(* IEC 61131-3 sources: PLC/exercises, 9 files *)

(* ---- practice_10.st ---- *)
(*
 * non revisonato
**)

PROGRAM _INIT

END_PROGRAM

PROGRAM _CYCLIC

    VAR
        start_button := "ingresso_1";
        stop_button := "ingresso_2";
        sensore_imbuto_alto := "ingresso_3";                 // Sensore parte alta dell'imbuto
        sensore_imbuto_basso := "ingresso_4";                // Sensore parte bassa dell'imbuto

        "uscita_1" := cilindro_valvola_ingersso_imbuto;      // Per rempimento imbuto
        "uscita_2" := cilindro_valvola_uscita_imbuto;        // Per svutamento imbuto
        "uscita_2" := motore_nasto_trasportatore;
        "uscita_2" := forno_cottura;

    END_VAR

    IF start_button AND NOT stop_button THEN
        start_ciclo.sensore_imbuto_basso := sensore_imbuto_basso;
        start_ciclo.sensore_imbuto_basso := sensore_imbuto_basso;
        start_ciclo.cilindro_valvola_ingersso_imbuto := cilindro_valvola_uscita_imbuto;
        start_ciclo.cilindro_valvola_uscita_imbuto := cilindro_valvola_uscita_imbuto;
        start_ciclo.motore_nasto_trasportatore := motore_nasto_trasportatore;
        start_ciclo.forno_cottura := forno_cottura;
        start_ciclo();
    ELSIF stop_button AND NOT start_button THEN
        stop_ciclo.cilindro_valvola_ingersso_imbuto := cilindro_valvola_uscita_imbuto;
        stop_ciclo.cilindro_valvola_uscita_imbuto := cilindro_valvola_uscita_imbuto;
        stop_ciclo.motore_nasto_trasportatore := motore_nasto_trasportatore;
        stop_ciclo.forno_cottura := forno_cottura;
        stop_ciclo();
    END_IF;

    FUNCTION_BLOCK start_ciclo
        (*
         * Avvia il ciclo produttivo del forno
        **)
        VAR_INPUT
            sensore_imbuto_alto: BOOL;
            sensore_imbuto_basso: BOOL;

            cilindro_valvola_ingersso_imbuto: BOOL;
            cilindro_valvola_uscita_imbuto: BOOL;
            motore_nasto_trasportatore: BOOL;
            forno_cottura: BOOL;
        END_VAR
        VAR
            fase := 0;
            timer_nastro := 0;
            timer_forno := 0;
        END_VAR

        IF sistem_bit_1sec AND motore_nasto_trasportatore THEN
            timer_nastro := timer_nastro + 1;
        ELSIF sistem_bit_1sec AND forno_cottura THEN
            timer_forno := timer_forno + 1;
        END_IF;

        CASE fase OF
            0:
                (*
                 * Controllo riempimento/svuotamento imbuto
                 *
                 * Entry point
                **)
                IF NOT sensore_imbuto_alto AND NOT sensore_imbuto_basso THEN
                    cilindro_valvola_uscita_imbuto := 0;
                    cilindro_valvola_ingersso_imbuto := 1;
                ELSIF sensore_imbuto_alto AND sensore_imbuto_basso THEN
                    cilindro_valvola_ingersso_imbuto := 0;
                    cilindro_valvola_uscita_imbuto := 1;
                    fase := 10;
                END_IF;

            10:
                (*
                 * Avvio e arresto nastro trasportatore per ingresso forno
                 *
                 * Entrata → fase 0 (riempimento/svuotamento imbuto)
                 * Uscita → fase 20 (forno cottura)
                **)
                IF NOT motore_nasto_trasportatore AND timer_nastro == 0 THEN
                    motore_nasto_trasportatore := 1;
                ELSIF motore_nasto_trasportatore AND timer_nastro == 15 THEN
                    motore_nasto_trasportatore := 0;
                    timer_nastro := 0;
                    fase := 20;
                END_IF;

            20:
                (*
                 * Accensione e spegnimento forno cottura
                 *
                 * Entrata → fase 20 (nastro trasportatore per ingresso forno)
                 * Uscita → fase 30 (nastro trasportatore per uscita forno)
                **)
                IF NOT forno_cottura THEN
                    forno_cottura := 1;
                ELSIF forno_cottura AND timer_forno == 10 THEN
                    forno_cottura := 0;
                    timer_forno := 0;
                    fase := 30;
                END_IF;

            30:
                (*
                 * Avvio e arresto nastro trasportatore per uscita forno
                 *
                 * Entrata → fase 30 (forno cottura)
                 * Uscita → fase 0 (riempimento/svuotamento imbuto)
                **)
                IF NOT motore_nasto_trasportatore THEN
                    motore_nasto_trasportatore := 1;
                ELSIF motore_nasto_trasportatore AND timer_nastro == 10 THEN
                    motore_nasto_trasportatore := 0;
                    timer_nastro := 0;
                    fase := 0;
                END_IF;

        END_CASE;

    END_FUNCTION_BLOCK

    FUNCTION_BLOCK stop_ciclo
        (*
         * Ferma il ciclo produttivo del forno
        **)
        VAR_INPUT
            cilindro_valvola_ingersso_imbuto: BOOL;
            cilindro_valvola_uscita_imbuto: BOOL;
            motore_nasto_trasportatore: BOOL;
            forno_cottura: BOOL;
        END_VAR

            cilindro_valvola_ingersso_imbuto := 0;
            cilindro_valvola_uscita_imbuto := 0;
            motore_nasto_trasportatore =: 0;
            forno_cottura := 0;

    END_FUNCTION_BLOCK

END_PROGRAM

PROGRAM _EXIT

END_PROGRAM

(* ---- practice_14.st ---- *)
(*
 * non revisionato
**)

PROGRAM _INIT

END_PROGRAM

PROGRAM _CYCLIC

    VAR
        A := "ingresso_1";
        B := "ingresso_2";
        conteggio : INT := 0;
    END_VAR

    contatore.A := A;
    contatore.B := B;
    contatore.conteggio := conteggio;
    contatore();

    FUNCTION_BLOCK contatore
        VAR_INPUT
            A : BOOL;
            B : BOOL;
            conteggio : INT;
        END_VAR
        VAR
            orario: BOOL := 0;
        END_VAR

        CASE fase OF
        0:
            IF NOT A AND NOT B THEN
                fase := 10;
            END_IF;
        10:
            IF A XOR B THEN
                IF A AND NOT B THEN
                    orario := 1;
                ELSIF NOT A AND B THEN
                    orario := 0;
                END_IF;
                fase := 20;
            END_IF;
        20:
            IF A AND B THEN
                fase := 30;
            END_IF;
        30:
            IF A XOR B THEN
                fase := 40;
            END_IF;
        40:
            IF orario THEN
                conteggio := conteggio + 1;
            ELSE
                conteggio := conteggio - 1;
            END_IF;
            fase := 0;

    END_FUNCTION_BLOCK

END_PROGRAM

PROGRAM _EXIT

END_PROGRAM

(* ---- practice_15.st ---- *)
(*
 * non revisionato
**)

PROGRAM _INIT

END_PROGRAM

PROGRAM _CYCLIC

    VAR
        A := "ingresso_1";
        B := "ingresso_2";
        preset := "ingresso_3";
        conteggio : INT := 0;
        orario: BOOL := 0;
        "uscita_4" := trasporto;
    END_VAR

    contatore.A := A;
    contatore.B := B;
    contatore.conteggio := conteggio;
    contatore();

    IF preset THEN
        contatore.conteggio := 0;
    END_IF;

    IF contatore.conteggio MOD 1000 == 0 THEN
        trasporto := 1;
    END_IF;

    FUNCTION_BLOCK contatore
        VAR_INPUT
            A : BOOL;
            B : BOOL;
            conteggio : INT;
        END_VAR
        VAR
            orario: BOOL := 0;
        END_VAR

        CASE fase OF
        0:
            IF NOT A AND NOT B THEN
                fase := 10;
            END_IF;
        10:
            IF A XOR B THEN
                IF A AND NOT B THEN
                    orario := 1;
                ELSIF NOT A AND B THEN
                    orario := 0;
                END_IF;
                fase := 20;
            END_IF;
        20:
            IF A AND B THEN
                fase := 30;
            END_IF;
        30:
            IF A XOR B THEN
                fase := 40;
            END_IF;
        40:
            IF orario THEN
                conteggio := conteggio + 1;
            ELSE
                conteggio := conteggio - 1;
            END_IF;
            fase := 0;

    END_FUNCTION_BLOCK

END_PROGRAM

PROGRAM _EXIT

END_PROGRAM

(* ---- practice_16.st ---- *)
(*
 * non revisionato
**)

PROGRAM _INIT

END_PROGRAM

PROGRAM _CYCLIC

    VAR
        A := "ingresso_1";
        B := "ingresso_2";
        reset := "ingresso_3";

        conteggio : INT := 0;

        "uscita_1" := led[0];
        "uscita_2" := led[1];
        "uscita_3" := led[2];
        "uscita_4" := led[3];
        "uscita_5" := led[4];
        "uscita_6" := led[5];
        "uscita_7" := led[6];
        "uscita_8" := led[7];
        "uscita_9" := led[8];
        "uscita_10" := led[9];
    END_VAR

    contatore.A := A;
    contatore.B := B;
    contatore.conteggio := conteggio;
    contatore();

    IF contatore.conteggio MOD 100 THEN
        FOR x := 0 TO conteggio BY 100 DO
            led[x] := 0;
        END_FOR;
    END_IF;

    IF reset OR contatore.conteggio MOD 2000 == 0 THEN
        FOR x := 0 TO 9 DO
           led[x] := 0;
        END_FOR;
    END_IF;

    FUNCTION_BLOCK contatore
        VAR_INPUT
            A : BOOL;
            B : BOOL;
            conteggio : INT;
        END_VAR
        VAR
            orario: BOOL := 0;
        END_VAR

        CASE fase OF
        0:
            IF NOT A AND NOT B THEN
                fase := 10;
            END_IF;
        10:
            IF A XOR B THEN
                IF A AND NOT B THEN
                    orario := 1;
                ELSIF NOT A AND B THEN
                    orario := 0;
                END_IF;
                fase := 20;
            END_IF;
        20:
            IF A AND B THEN
                fase := 30;
            END_IF;
        30:
            IF A XOR B THEN
                fase := 40;
            END_IF;
        40:
            IF orario THEN
                conteggio := conteggio + 1;
            ELSE
                conteggio := conteggio - 1;
            END_IF;
            fase := 0;

    END_FUNCTION_BLOCK

END_PROGRAM

PROGRAM _EXIT

END_PROGRAM

(* ---- practice_01.st ---- *)
(*
    EXERCISE 01

    Author: Chiliano Arcarese
    Revised by IVAN
*)

PROGRAM _INIT

END_PROGRAM

PROGRAM _CYCLIC

    VAR
        ingresso_rele := "ingresso_1";
        "uscita_1" := uscita_motore;
    END_VAR

    IF ingresso_rele AND uscita_motore THEN
        uscita_motore := 0;
    END_IF;

END_PROGRAM

PROGRAM _EXIT

END_PROGRAM

(* ---- practice_09.st ---- *)
(*
 * es 09
 * revisionato.
**)

PROGRAM _INIT
END_PROGRAM

PROGRAM _CYCLIC

    VAR

        (*
         *  >>>>>>>>>>>>>> !-NOTA-BENE-! <<<<<<<<<<<<<<<
         *
         *  I PIANI SONO NOMINATI COME 1°, 2° E 3.
         *  IL PIANO TERRA CORRISPONDE AL 1° PIANO.
         *
         *  >>>>>>>>>>>>>> !-NOTA-BENE-! <<<<<<<<<<<<<<<
        **)

        // Contesto relativo al 1 piano dell'edificio
        "uscita_1" := led_piano_1;                       // LED di segnalazione movimento cabina (1 == movimento)
        pulsante_chiamata_piano_1 := "ingresso_1";       // Pulsante di chiamata della cabina
        sensore_arrivo_piano_1 := "ingresso_2";          // Sensore di arrivo della cabina (1 == cabina presente)

        // Contesto relativo al 2 piano dell'edificio
        "uscita_2" := led_piano_2;
        pulsante_chiamata_piano_2 := "ingresso_3";
        sensore_arrivo_piano_2 := "ingresso_4";

        // Contesto relativo al 3 piano dell'edificio
        "uscita_3" := led_piano_3;
        pulsante_chiamata_piano_3 := "ingresso_5";
        sensore_arrivo_piano_3 := "ingresso_6";

        // Contesto interno alla cabina dell'ascensore
        pulsante_cabina_piano_1 := "ingresso_7";           //
        pulsante_cabina_piano_2 := "ingresso_8";           // Pulsante destinazione cabina
        pulsante_cabina_piano_3 := "ingresso_9";           //
        sensore_chiusura_porte := "ingresso_10";           // Sensore chiusura porte (1 == chiuse)
        pulsante_allarme := "ingresso_11";                 // Pulsante di emergenza, attiva un allarme di 20s
        allarme_cabina := "uscita_8";

        // Contesto motori cabina
        "uscita_4" := motore_up;
        "uscita_5" := motore_down;

        // Contesto motori porte
        "uscita_6" := motore_porte_open;
        "uscita_7" := motore_porte_close;

        timer: INT := 0;
        timer_porta: INT := 0;

    END_VAR

    (*
     * Inizializzazione variabili funzione `movimento_cabina`
    **)
    // Led movimento cabina
    movimento_cabina.led_piano_1 := led_piano_1;
    movimento_cabina.led_piano_2 := led_piano_2;
    movimento_cabina.led_piano_3 := led_piano_3;
    // Sensori presenza cabina
    movimento_cabina.sensore_arrivo_piano_1 := sensore_arrivo_piano_1;
    movimento_cabina.sensore_arrivo_piano_2 := sensore_arrivo_piano_2;
    movimento_cabina.sensore_arrivo_piano_3 := sensore_arrivo_piano_3;
     // Porte cabina
    movimento_cabina.sensore_chiusura_porte := sensore_chiusura_porte;
    movimento_cabina.motore_porte_open := motore_porte_open;
    // Motori cabina
    movimento_cabina.motore_up := motore_up;
    movimento_cabina.motore_down := motore_down;

    (*
     * Chiamata della cabina da uno dei piani presenti.
    **)
    IF pulsante_chiamata_piano_1 THEN
        movimento_cabina.chiamta_esterna := TRUE;
        movimento_cabina.pulsante_chiamata := pulsante_chiamata_piano_1;
        movimento_cabina.piano_chiamata := 1;
        movimento_cabina();
    ELSIF pulsante_chiamata_piano_2 THEN
        movimento_cabina.chiamta_esterna := TRUE;
        movimento_cabina.pulsante_chiamata := pulsante_chiamata_piano_2;
        movimento_cabina.piano_chiamata := 2;
        movimento_cabina();
    ELSIF pulsante_chiamata_piano_3 THEN
        movimento_cabina.chiamta_esterna := TRUE;
        movimento_cabina.pulsante_chiamata := pulsante_chiamata_piano_3;
        movimento_cabina.piano_chiamata := 3;
        movimento_cabina();
    END_IF;

    (*
     * Risposta della cabina da pulsante interno.
    **)
    IF pulsante_cabina_piano_1 AND NOT sensore_arrivo_piano_1 THEN
        movimento_cabina.chiamta_esterna := FALSE;
        movimento_cabina.pulsante_chiamata := pulsante_cabina_piano_1;
        movimento_cabina.piano_chiamata := 1;
        movimento_cabina();
    ELSIF pulsante_cabina_piano_2 AND NOT sensore_arrivo_piano_2 THEN
        movimento_cabina.chiamta_esterna := FALSE;
        movimento_cabina.pulsante_chiamata := pulsante_cabina_piano_2;
        movimento_cabina.piano_chiamata := 2;
        movimento_cabina();
    ELSIF pulsante_cabina_piano_3 AND NOT sensore_arrivo_piano_3 THEN
        movimento_cabina.chiamta_esterna := FALSE;
        movimento_cabina.pulsante_chiamata := pulsante_cabina_piano_3;
        movimento_cabina.piano_chiamata := 3;
        movimento_cabina();
    END_IF;

    IF pulsante_allarme THEN
        allarme_cabina := 1;
        timer := 0;
    END_IF;

    IF sistem_bit_1sec THEN
        timer := timer + 1;
    END_IF;

    IF sistem_bit_1sec AND NOT sensore_chiusura_porte THEN
        timer_porta := timer_porta + 1;
    END_IF;

    IF timer == 20 AND allarme_cabina THEN
        allarme_cabina := 0;
        timer := 0;
    END_IF;

    // Chiusura porta ascensore automatica dopo 40 sec
    IF timer_porta > 40 AND NOT sensore_chiusura_porte AND NOT motore_porte_close THEN
        timer_porta := 0;
        motore_porte_close := 1;
    ELSIF sensore_chiusura_porte AND motore_porte_close THEN
        motore_porte_close := 0;
    END_IF;
 THEN

    FUNCTION_BLOCK movimento_cabina
    (*
     * Muove la cabina sui piani in base agli input dei pulsanti presenti in ogni piano.
    **)

        VAR_INPUT
            piano_chiamata: INT;
            chiamta_esterna: BOOL;
            pulsante_chiamata: BOOL;            // Pulsante di chiamata della cabina
            led_piano_1: BOOL;
            led_piano_2: BOOL;
            led_piano_3: BOOL;

            // Sensori presenza cabina
            sensore_arrivo_piano_1: BOOL;
            sensore_arrivo_piano_2: BOOL;
            sensore_arrivo_piano_3: BOOL;

            // Porte cabina
            sensore_chiusura_porte: BOOL;
            motore_porte_open: BOOL;

            // Motori cabina
            motore_up: BOOL;
            motore_down: BOOL;
        END_VAR

        VAR
            fase: INT := 0;                     // Variabile locale per i casi del CASE OF
        END_VAR

        IF pulsante_chiamata_piano AND NOT led_piano_1 AND NOT led_piano_2 AND NOT led_piano_3 THEN
            // Segnalo cabina in uso su tutti i piani
            led_piano_1 := TRUE;
            led_piano_2 := TRUE;
            led_piano_3 := TRUE;

            CASE fase OF

                0:
                    (*
                     * Localizzazione della cabina fra i piani e reindirizzamento verso il piano di chiamata.
                     *
                     * Entrate → Case entry point
                     *
                     * Uscite  → Spostamenti cabina (30, 40, 50)
                     *           Apertura porte (10)
                    **)
                    IF sensore_arrivo_piano_1 AND NOT sensore_arrivo_piano_2 AND NOT sensore_arrivo_piano_3 THEN
                        // Chiamata da piano
                        IF piano_chiamata == 1 AND chiamta_esterna THEN
                            fase := 10;
                        ELSIF piano_chiamata == 2 AND chiamta_esterna THEN
                            fase := 50;
                        ELSIF piano_chiamata == 3 AND chiamta_esterna THEN
                            fase := 40;
                        // Chiamata da cabina
                        ELSIF piano_chiamata == 1 AND NOT chiamta_esterna THEN
                            fase := 0;
                        ELSIF piano_chiamata == 2 AND NOT chiamta_esterna THEN
                            fase := 20;
                        ELSIF piano_chiamata == 3 AND NOT chiamta_esterna THEN
                            fase := 20;
                        END_IF;
                    ELSIF NOT sensore_arrivo_piano_1 AND sensore_arrivo_piano_2 AND NOT sensore_arrivo_piano_3 THEN
                        // Chiamata da piano
                        IF piano_chiamata == 1 AND chiamta_esterna THEN
                            fase := 30;
                        ELSIF piano_chiamata == 2 AND chiamta_esterna THEN
                            fase := 10;
                        ELSIF piano_chiamata == 3 AND chiamta_esterna THEN
                            fase := 40;
                        // Chiamata da cabina
                        ELSIF piano_chiamata == 1 AND NOT chiamta_esterna THEN
                            fase := 0;
                        ELSIF piano_chiamata == 2 AND NOT chiamta_esterna THEN
                            fase := 20;
                        ELSIF piano_chiamata == 3 AND NOT chiamta_esterna THEN
                            fase := 20;
                        END_IF;
                    ELSIF NOT sensore_arrivo_piano_1 AND NOT sensore_arrivo_piano_2 AND sensore_arrivo_piano_3 THEN
                        // Chiamata da piano
                        IF piano_chiamata == 1 AND chiamta_esterna THEN
                            fase := 30;
                        ELSIF piano_chiamata == 2 AND chiamta_esterna THEN
                            fase := 50;
                        ELSIF piano_chiamata == 3 AND chiamta_esterna THEN
                            fase := 10;
                        // Chiamata da cabina
                        ELSIF piano_chiamata == 1 AND NOT chiamta_esterna THEN
                            fase := 0;
                        ELSIF piano_chiamata == 2 AND NOT chiamta_esterna THEN
                            fase := 20;
                        ELSIF piano_chiamata == 3 AND NOT chiamta_esterna THEN
                            fase := 20;
                        END_IF;
                    END_IF;

                10:
                    (*
                     * Apertura porte cabina.
                     *
                     * Entrata → Localizzazione e reindirizzamento (0)
                    **)
                    IF sensore_chiusura_porte AND NOT motore_porte_open THEN
                        motore_porte_open := 1;
                    ELSIF NOT sensore_chiusura_porte AND motore_porte_open THEN
                        motore_porte_open := 0;
                    END_IF;
                    fase := 0;

                20:
                    (*
                     * Chiusura porte cabina.
                     *
                     * Entrata → Localizzazione e reindirizzamento (0)
                    **)
                    IF NOT sensore_chiusura_porte AND NOT motore_porte_close THEN
                        motore_porte_close := 1;
                    ELSIF sensore_chiusura_porte AND motore_porte_close THEN
                        motore_porte_close := 0;
                    END_IF;
                    fase := 0;
                    // In fase 0 il movimento viene poi gestito come una chiamata a piano ma pertendo a porte chiuse
                    chiamta_esterna := TRUE;

                30:
                    (*
                     * Spostamento cabina verso il 1° piano.
                     *
                     * Entrata → Localizzazione e reindirizzamento (0)
                     *
                     * Uscita → Apertura porte (10)
                    **)
                    IF NOT motore_up AND NOT motore_down AND sensore_chiusura_porte THEN
                        motore_down := 1;
                    ELSIF NOT motore_up AND motore_down AND sensore_arrivo_piano_1 THEN
                        motore_down := 0;
                        fase := 10;
                    ELSIF motore_up OR motore_down AND NOT sensore_chiusura_porte THEN
                        // ALLARME PORTA CABINA APERTA
                    END_IF;

                40:
                    (*
                     * Spostamento cabina verso il 3° piano.
                     *
                     * Entrata → Localizzazione e reindirizzamento (0)
                     *
                     * Uscita → Apertura porte (10)
                    **)
                    IF NOT motore_up AND NOT motore_down AND sensore_chiusura_porte THEN
                        motore_up := 1;
                    ELSIF motore_up AND NOT motore_down AND sensore_arrivo_piano_3 THEN
                        motore_up := 0;
                        fase := 10;
                    ELSIF motore_up OR motore_down AND NOT sensore_chiusura_porte THEN
                        // ALLARME PORTA CABINA APERTA
                    END_IF;

                50:
                    (*
                     * Spostamento cabina verso il 2° piano. La cabina si sporterà a partire dal basso o dall'alto.
                     *
                     * Entrata → Localizzazione e reindirizzamento (0)
                     *
                     * Uscita → Apertura porte (10)
                    **)
                    IF NOT motore_up AND NOT motore_down THEN
                        IF sensore_arrivo_piano_3 AND NOT sensore_arrivo_piano_1 AND NOT sensore_arrivo_piano_2 THEN
                            motore_down := 1;
                        ELSIF sensore_arrivo_piano_1 AND NOT sensore_arrivo_piano_2 AND NOT sensore_arrivo_piano_3 THEN
                            motore_up := 1;
                        END_IF;
                    ELSIF motore_down AND NOT motore_up THEN
                        IF sensore_arrivo_piano_2 THEN
                            motore_down := 0;
                            fase := 10;
                        END_IF;
                    ELSIF NOT motore_down AND motore_up THEN
                        IF sensore_arrivo_piano_2 THEN
                            motore_up := 0;
                            fase := 10;
                        END_IF;

            END_CASE;

        END_IF;

    END_FUNCTION_BLOCK

END_PROGRAM

PROGRAM _EXIT
END_PROGRAM

(* ---- practice_11.st ---- *)
(*
 * non revisionato
**)

PROGRAM _INIT

END_PROGRAM

PROGRAM _CYCLIC

    VAR
        rele[0] := "ingresso_1"
        rele[1] := "ingresso_2"
        rele[2] := "ingresso_3"
        rele[3] := "ingresso_4"
        rele[4] := "ingresso_5"
        rele[6] := "ingresso_6"
        rele[7] := "ingresso_7"
        rele[8] := "ingresso_8"
        rele[9] := "ingresso_9"
        rele[10] := "ingresso_10"

        "uscita_1" := motori[0];
        "uscita_2" := motori[1];
        "uscita_3" := motori[2];
        "uscita_4" := motori[3];
        "uscita_5" := motori[4];
        "uscita_6" := motori[5];
        "uscita_7" := motori[6];
        "uscita_8" := motori[7];
        "uscita_9" := motori[8];
        "uscita_10" := motori[9];
    END_VAR

    FOR x := 0 TO 9 BY 1 DO
        IF rele[0] THEN
            motori[x] := 0;
        ELSE
            motori[x] := 1;
        END_IF;
    END_FOR;

END_PROGRAM

PROGRAM _EXIT

END_PROGRAM

(* ---- practice_12.st ---- *)
(*
 * non revisionato
**)

PROGRAM _INIT

END_PROGRAM

PROGRAM _CYCLIC

    VAR
        pulsante := "ingresso_1";
        "uscita_1" := led[0]
        "uscita_2" := led[1]
        "uscita_3" := led[2]
        "uscita_4" := led[3]
        "uscita_5" := led[4]
        "uscita_6" := led[5]
        "uscita_7" := led[6]
        "uscita_8" := led[7]
        "uscita_9" := led[8]
        "uscita_10" := led[9]
        fase : INT := 0;
    END_VAR

    IF pulsante THEN
        CASE fase OF
            0:
                led[fase] := 1;
                fase := fase + 1;
            1:
                led[fase] := 1;
                fase := fase + 1;
            2:
                led[fase] := 1;
                fase := fase + 1;
            3:
                led[fase] := 1;
                fase := fase + 1;
            4:
                led[fase] := 1;
                fase := fase + 1;
            5:
                led[fase] := 1;
                fase := fase + 1;
            6:
                led[fase] := 1;
                fase := fase + 1;
            7:
                led[fase] := 1;
                fase := fase + 1;
            8:
                led[fase] := 1;
                fase := fase + 1;
            9:
                led[fase] := 1;
                fase := fase + 1;
            10:
                FOR x := 0 TO 9 DO
                    led[x] := 0;
                END_FOR;
                fase := 0;

        END_CASE;

END_PROGRAM

PROGRAM _EXIT

END_PROGRAM

(* ---- practice_17.st ---- *)
(*
 * non revisionato
**)

PROGRAM _INIT

END_PROGRAM

PROGRAM _CYCLIC

    VAR
        pulsante_carico_ricetta := "ingresso_1";
        finecorsa_passo         := "ingresso_2";
        ricetta : ARRAY[0..10]  := "ingresso_3";

        nr_posizione : INT := 0;
        posizione;
        appoggio1;
        appoggio2;

        mappa : ARRAY[0..10] OF ARRAY[1..10] := [
            pos_1 : ARRAY[0..10] OF INT, pos_2 : ARRAY[0..10] OF INT, pos_3 : ARRAY[0..10] OF INT,
            pos_4 : ARRAY[0..10] OF INT, pos_5 : ARRAY[0..10] OF INT, pos_6 : ARRAY[0..10] OF INT,
            pos_7 : ARRAY[0..10] OF INT, pos_8 : ARRAY[0..10] OF INT, pos_9 : ARRAY[0..10] OF INT,
            pos_10 : ARRAY[0..10] OF INT
        ];
    END_VAR

    IF nr_posizione >= 10 THEN
        nr_posizione := 0;
    END_IF;

    prima_colonna_vuota.col1 := mappa[nr_posizione];

    IF pulsante_carico_ricetta AND prima_colonna_vuota() THEN
        // Scrive nella prima colonna
        scrivi_colonna.colonna_vuota := mappa[0];
        scrivi_colonna.ricetta := ricetta;
        scrivi_colonna();
        nr_posizione := nr_posizione + 1;       // Sposto l'offset sulla prossima colonna libera

    ELSIF pulsante_carico_ricetta AND NOT prima_colonna_vuota() THEN
        // Scala le colonne di 1
        posizione := nr_posizione;
        IF posizione >= 2 THEN
            FOR i := 0 TO nr_posizione DO
                appoggio1 := mappa[posizione];
                appoggio2 := mappa[posizione - 1];
                FOR x := 0 TO 10 DO
                    appoggio1[x] := appoggio2[x];
                END_FOR;
                posizione := posizione - 1;
            END_FOR;
        END_IF;

        // scive la nuova ricetta nella 1a colonna
        scrivi_colonna.colonna_vuota := mappa[0];
        scrivi_colonna();
        nr_posizione := nr_posizione + 1;
    END_IF;

    FUNCTION prima_colonna_vuota : BOOL
        (*
         * Ritorna 1 se la l'array ricevuto in input è vuoto
        **)
        VAR_INPUT
            col1: ARRAY[1..10] OF INT;
        END_VAR

        VAR
            vuota : BOOL := 1;
        END_VAR

        FOR i := 0 TO 10 DO
            IF col1[i] == 0 THEN
                vuota := 0;
            END_IF;
        END_FOR;
        RETURN vuota;
    END_FUNCTION

    FUNCTION scrivi_colonna : INT
        (*
         * Copia un array su un'altro array
        **)
        VAR_INPUT
            colonna_vuota : ARRAY[1..10] OF INT;
            ricetta : ARRAY[1..10] OF INT;
        END_VAR

        FOR x := 0 TO 10 DO
            colonna_vuota[x] := ricetta[x];
        END_FOR;
        RETURN 1;
    END_FUNCTION

END_PROGRAM

PROGRAM _EXIT

END_PROGRAM
